(* CODESYS project mobject-vision-nodepack.library
   Company: mobject
   DefaultNamespace: mobject-vision-nodepack
   Version: 0.1.0
   Placeholder: mobject-vision-nodepack
   Author: mobject dev team
   Title: mobject-vision-nodepack

Project tree, tasks and I/O mapping:
  libraries: mobject-graph, 0.3.0 (mobject); mobject-vision-datatypes, 0.1.0 (mobject)
  function block VisionNodePack [ST]: RegisterWithNodeFactory
*)

// VisionNodePack
{attribute 'linkalways'} 
{attribute 'no_explicit_call' := 'This FB is a CLASS and must be accessed using methods or properties'}
{attribute 'enable_dynamic_creation'}
FUNCTION_BLOCK VisionNodePack IMPLEMENTS I_NodePack
VAR
	//node : Node;
END_VAR

METHOD PUBLIC RegisterWithNodeFactory
VAR_INPUT
	NodeFactory : I_NodeFactory;
END_VAR
//NodeFactory.AddNodeAsPrototype('Vision/Node',Node);
END_METHOD

END_FUNCTION_BLOCK
